{attribute 'linkalways'} 
{attribute 'no_explicit_call' := 'This FB is a CLASS and must be accessed using methods or properties'}
{attribute 'enable_dynamic_creation'}
FUNCTION_BLOCK _ETcVnPaddingMode EXTENDS EnumDatatypeBase
VAR
	localData : ETcVnPaddingMode;
	activeData : REFERENCE TO ETcVnPaddingMode;
	enumBaseDatatype : _DINT(localData);
END_VAR

METHOD PRIVATE AddLocalEnumeration
VAR_INPUT
	Enumeration : T_MAXSTRING;
	Value : ETcVnPaddingMode;
END_VAR
AddEnumeration(Enumeration, Value);
END_METHOD

PROPERTY PUBLIC Address : PVOID
GET
Address := ADR(activeData);
END_GET
END_PROPERTY

METHOD PUBLIC ClearReference
VAR_INPUT
END_VAR
activeData REF= localData;
SetBaseDatatypeReference();
END_METHOD

METHOD PUBLIC Clone : I_Datatype
VAR
    pClone : POINTER TO _ETcVnPaddingMode;
END_VAR
pClone := __NEW(_ETcVnPaddingMode(InitialValue := Value));
Clone := pClone^;
END_METHOD

METHOD FB_init : BOOL
VAR_INPUT
	bInitRetains : BOOL; // if TRUE, the retain variables are initialized (warm start / cold start)
	bInCopyCode : BOOL;  // if TRUE, the instance afterwards gets moved into the copy code (online change)
	InitialValue : ETcVnPaddingMode;
END_VAR
localData := InitialValue;
AddBaseDatatype(enumBaseDatatype);
ClearReference();

AddLocalEnumeration('TCVN_PM_NONE', ETcVnPaddingMode.TCVN_PM_NONE);
AddLocalEnumeration('TCVN_PM_CROP_CENTER', ETcVnPaddingMode.TCVN_PM_CROP_CENTER);
AddLocalEnumeration('TCVN_PM_LETTERBOX', ETcVnPaddingMode.TCVN_PM_LETTERBOX);
END_METHOD

PROPERTY PUBLIC Identifier : T_MAXSTRING
GET
Identifier := 'ETcVnPaddingMode';
END_GET
END_PROPERTY

METHOD IsEnumeratorValueEqual : BOOL
VAR_INPUT
	Enumerator : I_KeyValueForwardEnumerator;
END_VAR
VAR
	storedValue : ETcVnPaddingMode;
END_VAR
IF NOT Enumerator.TryGet(storedValue) THEN
	RETURN;
END_IF

IsEnumeratorValueEqual := storedValue = activeData;
END_METHOD

METHOD PUBLIC MakeReferenceTo
VAR_INPUT
	ReferenceTarget : REFERENCE TO ETcVnPaddingMode;
END_VAR
activeData REF= ReferenceTarget;
SetBaseDatatypeReference();
END_METHOD

METHOD PROTECTED SetBaseDatatypeReference
VAR_INPUT
END_VAR
enumBaseDatatype.MakeReferenceTo(activeData);
END_METHOD

PROPERTY PUBLIC Size : UDINT
GET
Size := SIZEOF(activeData);
END_GET
END_PROPERTY

METHOD TryMakeReferenceTo : BOOL
VAR_INPUT
	Target : I_Datatype;
END_VAR
VAR
	targetAsEnum : I_EnumDatatype;
	pTargetData : POINTER TO ETcVnPaddingMode;
END_VAR
IF NOT Target.TryResolveAsEnumDatatype(targetAsEnum) THEN
	RETURN;
END_IF

IF targetAsEnum.Identifier <> Identifier THEN
	RETURN;
END_IF

pTargetData := Target.Address;
activeData REF= pTargetData^;
SetBaseDatatypeReference();
TryMakeReferenceTo := TRUE;
END_METHOD

PROPERTY PUBLIC Value : ETcVnPaddingMode
GET
Value := activeData;
END_GET
SET
activeData := Value;
END_SET
END_PROPERTY

END_FUNCTION_BLOCK

(* stored: Version 1.1.0.1
   POU _ETcVnPaddingMode: Id {00e296e8-ee2b-4a09-9709-7e044ec0ab43}, SpecialFunc None
   Folder Constructor: Id {146c51eb-637d-432b-b85c-5f12010ff1b5}
   Folder Private: Id {7ddc75bc-781d-4133-8a72-ad29258bdf8f}
   Folder Protected: Id {884f16c3-4c9c-4a57-b76b-6203564a616f}
   Method AddLocalEnumeration: Id {d84fa774-2bf1-4088-aa68-5c843d4e5f7f}
   Property Address: Id {38322df8-b04a-4438-bcfb-2829538f85ab}
   Get Get: Id {c61e8f8c-7d02-48f3-a1c2-c0011cbd027d}
   Method ClearReference: Id {0bbc73fb-a7f7-490f-917c-d4e856ff1868}
   Method Clone: Id {f4a024c0-0566-47e2-a515-078b8dd28bc3}
   Method FB_init: Id {85da4cd3-f7fa-4f20-8de6-865c45852f94}
   Property Identifier: Id {d8659d90-6b74-4222-af56-e189514db259}
   Get Get: Id {60f9e646-0b6a-4cba-973c-f80a00139f7f}
   Method IsEnumeratorValueEqual: Id {882e331b-3022-448c-b168-0a85fd6c212f}
   Method MakeReferenceTo: Id {65fccf7e-4e58-4bf7-b4d0-e971aa5bdca8}
   Method SetBaseDatatypeReference: Id {fe195034-f999-4871-aeca-097ab5dda550}
   Property Size: Id {72289449-6841-4f7e-b888-ee2d94cbd084}
   Get Get: Id {6f1f40c5-e522-4458-8378-86add1986016}
   Method TryMakeReferenceTo: Id {3f69e9d7-bab8-4bb6-b184-a0fcdc72ad88}
   Property Value: Id {878926cc-efa7-4ee9-aa2d-18e29222a7b2}
   Get Get: Id {5cbd04d1-1adc-4297-a979-5a47e5eb2080}
   Set Set: Id {bf742784-a34a-42b7-9233-b20ad1246ddc} *)
